(* PLC project  *)

CONFIGURATION Empty_Module_19
END_CONFIGURATION
